// Implicitly generated code : DO NOT EDIT
FUNCTION CheckDivLReal : LREAL
VAR_INPUT
	divisor:LREAL;
END_VAR

// Implicitly generated code : Only an Implementation suggestion
{noflow}
IF divisor = 0 THEN
	GVL_Checks.diCheckDivLReal := GVL_Checks.diCheckDivLReal +1;
	CheckDivLReal:=1;
ELSE
	CheckDivLReal:=divisor;
END_IF;
{flow}

END_FUNCTION

(* stored: Version 1.1.0.1, ProductVersion 3.1.4024.12
   POU CheckDivLReal: Id {47bbda28-7080-43c5-8916-26d93498efc2}, SpecialFunc CheckDivReal64 *)
